# EPICS autosave request: iocBoot/obsolete/ioc13MeasComp1208/auto_settings.req
file "USB1208_settings.req", P=13USB1208:
